// TIA Portal V21 export
DATA_BLOCK "DB622"   // DB622
TITLE = DB620
{ S7_Optimized_Access := 'FALSE' }
// CIP POPUPS
// stored: AutoNumber false
   VAR RETAIN
      NoCycleSelectedPopup : Bool;
      MainPopupMsg1 : Bool;
      MainPopupMsg2 : Bool;
   END_VAR
BEGIN
END_DATA_BLOCK
